FUNCTION_BLOCK Day1
VAR_INPUT
END_VAR
VAR_OUTPUT
END_VAR
VAR
END_VAR

END_FUNCTION_BLOCK

(* stored: Version 1.1.0.1, ProductVersion 3.1.4024.6
   POU Day1: Id {b71f8504-6820-4310-8889-ac39239075e1}, SpecialFunc None *)
